Staubli VAL3: txtBoxDyn.pgx

public program txtBoxDyn(string x_sMessage, num x_nRow, num x_nCol, num x_nBoxWidth)
  local num l_i
  local num l_nError
  local num l_nRow
  local num l_nCol
begin
  // This program displays a message on the MCP composed of a
  // static part and a dynamic part
  //
  // Input param
  // x_sMessage    : Message to display
  // x_nBoxWidth   : width of the message box to display
  //
  //
  // Created 23-02-05                           C.CURRIVAND
  //------------------------------------------------------------------
  //
  // Set default width if parameter is not consistent
  if x_nBoxWidth<=0
    x_nBoxWidth=5
  endIf
  //
  // Format the message to display (result is array of string called sWrkString[])
  // BoxWidth may be adjusted if one string is longer than boxWidth
  call setString(x_sMessage,x_nBoxWidth,l_nError)
  // Add an item to the working string array to reserve space for dynamic text
  insert(sWrkString[size(sWrkString)])
  x_nCol=roundDown((40-x_nBoxWidth)/2)
  //
  // display message Box
  nTxtBoxCol=x_nCol
  nTxtBoxRow=x_nRow
  nTxtBoxWidth=x_nBoxWidth-2
  call msgBoxDisplay(x_nBoxWidth)
  //
end
